INTERFACE ITcoContexBuilder

METHOD WithLogger : ITcoContexBuilder
VAR_INPUT
END_VAR
END_METHOD

END_INTERFACE

(* stored: Version 1.1.0.1, ProductVersion 3.1.4024.9
   Itf ITcoContexBuilder: Id {eab58bda-2fec-063c-131d-ae773937ca95}
   Method WithLogger: Id {abced830-4a55-0d4e-16ed-00d59a233b9a} *)
